// TIA Portal V16 export
// export: Created 2022-02-04T14:40:23.3671813Z, ExportSetting WithDefaults, DisplayName Totally Integrated Automation Portal, DisplayVersion V16 Update 1, DisplayName TIA Portal Version Control Interface, DisplayVersion V16, DisplayName TIA Portal Openness, DisplayVersion V16, DisplayName SINAMICS Startdrive Advanced, DisplayVersion V16 Update 5, DisplayName SINAMICS Startdrive G130, G150, S120, S150, SINAMICS MV, S210, DisplayVersion V16 Update 5, DisplayName SINAMICS Startdrive G110M, G120, G120C, G120D, G120P, G115D, DisplayVersion V16 Update 5, DisplayName STEP 7 Professional, DisplayVersion V16, DisplayName STEP 7 Safety, DisplayVersion V16, DisplayName WinCC Advanced, DisplayVersion V16, DisplayName SIMATIC Visualization Architect, DisplayVersion V16
DATA_BLOCK "DynamicLayer_CNTL_DB"   // DB24
AUTHOR : Aspir
VERSION : 0.1
// stored: AutoNumber true, InstanceOfName DynamicLayer_CNTL, InstanceOfType FB
"DynamicLayer_CNTL"
   // VAR_INPUT
   //    NewPack : Bool;
   //    EnableDynamicLayer : Bool;
   //    NotOkSensor : Bool;
   //    PackMaxHeight : Int;
   //    BoardsInLay : Int;
   //    BoardsInCurrentPack : Int;
   // END_VAR
   // VAR_OUTPUT
   //    ActualMaxHeight : Int;
   // END_VAR
   // VAR RETAIN
   //    NotOkSensor_old : Bool;
   //    notOk_Counter : Int;
   // END_VAR
BEGIN
END_DATA_BLOCK
